{attribute 'linkalways'} 
{attribute 'no_explicit_call' := 'This FB is a CLASS and must be accessed using methods or properties'}
{attribute 'enable_dynamic_creation'}
FUNCTION_BLOCK Node_F_VN_GetAt_SINT EXTENDS VisionNode
VAR
    ipContainer : _ITcVnContainer;
    nElement : _SINT(0);
    nIndex : _ULINT(0);
    hrPrev : _HRESULT(S_OK);
    hresult : _HRESULT(S_OK);
END_VAR

METHOD PUBLIC  Clone : I_Node
VAR
	pNode : POINTER TO Node_F_VN_GetAt_SINT;
END_VAR
pNode := __NEW(Node_F_VN_GetAt_SINT);
Clone := pNode^;
END_METHOD

METHOD FB_init : BOOL
VAR_INPUT
	bInitRetains : BOOL; // if TRUE, the retain variables are initialized (warm start / cold start)
	bInCopyCode : BOOL;  // if TRUE, the instance afterwards gets moved into the copy code (online change)
END_VAR
AddInput('ipContainer', ipContainer);
AddParameter('nIndex', nIndex);
AddInput('hrPrev', hrPrev);
AddOutput('nElement', nElement);
AddOutput('hresult',hresult);
END_METHOD

METHOD PROTECTED OnExecute
hresult.Value := F_VN_GetAt_SINT(
    ipContainer := ipContainer.Value,
    nElement := nElement.Value,
    nIndex := nIndex.Value,
    hrPrev:= hrPrev.Value);
END_METHOD

METHOD PUBLIC PreExecutionCheck
VAR_INPUT
	Check : I_PreExecutionChecks;
END_VAR
Check.IsTrue(ipContainer.IsValid, 'ipContainer must be a valid container');
Check.IsTrue(ipContainer.IsType(TC_GLOBAL_CONST_LIST.ContainerType_Vector_SINT), 'ipContainer contains incorrect type');
END_METHOD

END_FUNCTION_BLOCK

(* stored: Version 1.1.0.1, ProductVersion 3.1.4026.13
   POU Node_F_VN_GetAt_SINT: Id {bd208cd5-966d-4602-aa23-12f4390f7c78}, SpecialFunc None
   Folder Constructor: Id {a63bb5da-7abf-4c45-a89c-71aad42b12bb}
   Method Clone: Id {86d87d1d-73aa-48b8-bfe2-58e92b447053}
   Method FB_init: Id {305bece1-b3ee-4208-8455-26b79e22caa7}
   Method OnExecute: Id {807e2633-de6a-4fa2-aa23-0a464a2d863f}
   Method PreExecutionCheck: Id {a7e9e490-8f08-47f5-bffd-81e1d6fb82ec} *)
